(*
---Control step base interface
*)
FUNCTION_BLOCK ActStepBase IMPLEMENTS ITFActStep
VAR CONSTANT
	{attribute 'hide'}
	BEGIN_STEP		:DINT:=10;
	{attribute 'hide'}
	DONE_STEP		:DINT:=60000;
	{attribute 'hide'}
	ERR_DONE_STEP	:DINT:=65000;
	{attribute 'hide'}
	PAUSE_STEP		:DINT:=65500;
END_VAR
VAR_INPUT
END_VAR
VAR_OUTPUT
	step			:DINT;
	errStep			:DINT;
	pauseNextStep	:DINT;
END_VAR
VAR
	//{attribute 'hide'}
	actState		:ST_ActStep_State;
END_VAR

getStep();

(*
---Continue action
*)
METHOD Act_Continue : BOOL
VAR_INPUT
END_VAR
actState.paused:=FALSE;
actState.step:=actState.nextStep;
END_METHOD

(*
---Trigger action
*)
METHOD Act_Ex : BOOL
VAR_INPUT
END_VAR
IF NOT actState.busy AND NOT actState.error THEN
	Act_Ex:=actState.ex:=actState.busy:=TRUE;
ELSE
	Act_Ex:=FALSE;
END_IF
END_METHOD

(*
---Init all status
*)
METHOD Act_Init : BOOL
VAR_INPUT
END_VAR
actState.ex:=actState.pause:=actState.busy:=actState.done:=actState.error:=FALSE;
actState.step:=actState.errStep:=step:=0;
actState.errID:=0;
actState.errMsg:='';

Act_Init:=TRUE;
END_METHOD

(*
---Pause action
*)
METHOD Act_Pause : BOOL
VAR_INPUT
	pause:BOOL;
END_VAR
actState.pause:=pause;
Act_Pause:=TRUE;
END_METHOD

(*
---: add step;
---:
	nextStep: step 增量值;
	checkPause: 是否检测当前 pause; 如果 checkPause:=TRUE, 且暂停被触发后, 当前 step 暂停递增;
*)
METHOD addStep : DINT
VAR_INPUT
	nextStep			:DINT:=0;
	checkPause			:BOOL:=FALSE;// 检查是否暂停，暂停则不递增step
END_VAR
IF checkPause THEN
	IF NOT actState.pause THEN
		actState.step:=actState.step+nextStep;
	END_IF
ELSE
	actState.step:=actState.step+nextStep;
END_IF

addStep:=step:=actState.step;
END_METHOD

(*
---Get action state
*)
METHOD getActState : ST_ActStep_State
VAR_INPUT
END_VAR
getActState:=actState;
END_METHOD

(*
---Get error id
*)
METHOD getErrID : DINT
VAR_INPUT
END_VAR
getErrID:=actState.errID;
END_METHOD

(*
---Get error message
*)
METHOD getErrMsg : STRING(255)
VAR_INPUT
END_VAR
getErrMsg:=actState.errMsg;
END_METHOD

(*
---Get error step
*)
METHOD getErrStep : DINT
VAR_INPUT
END_VAR
getErrStep:=actState.errStep;
END_METHOD

(*
---Get step
*)
METHOD getStep : DINT
VAR_INPUT
END_VAR
getStep:=step:=actState.step;
END_METHOD

(*
---Check busy state
*)
METHOD isBusy : BOOL
VAR_INPUT
END_VAR

isBusy:=actState.busy;
END_METHOD

(*
---Check done state
*)
METHOD isDone : BOOL
VAR_INPUT
END_VAR

isDone:=actState.done;
END_METHOD

(*
---Check error state
*)
METHOD isError : BOOL
VAR_INPUT
END_VAR

isError:=actState.error;
END_METHOD

(*
---Check trigger state
*)
METHOD isEx : BOOL
VAR_INPUT
END_VAR

isEx:=actState.ex;
END_METHOD

(*
---Check pause state
*)
METHOD isPause : BOOL
VAR_INPUT
END_VAR

isPause:=actState.pause;
END_METHOD

(*
---Set busy flag
*)
METHOD setBusyFlag
VAR_INPUT
END_VAR
//actState.busy:=TRUE;
actState.ex:=actState.done:=actState.error:=FALSE;
actState.errID:=0;
actState.step:=step:=actState.errStep:=errStep:=actState.nextStep:=pauseNextStep:=0;
actState.errMsg:='';
END_METHOD

(*
---Set done flag
*)
METHOD setDoneFlag
VAR_INPUT
END_VAR
actState.busy:=FALSE;
actState.pause:=FALSE;
actState.done:=TRUE;
actState.error:=FALSE;
actState.errID:=0;
actState.errMsg:='';
END_METHOD

(*
---Set error done flag
*)
METHOD setErrDoneFlag
VAR_INPUT
END_VAR
actState.busy:=FALSE;
actState.pause:=FALSE;
actState.done:=FALSE;
actState.error:=TRUE;
END_METHOD

(*
---Set error id
*)
METHOD setErrID
VAR_INPUT
	errID:DINT;
END_VAR
actState.errID:=errID;
errStep:=actState.errStep:=actState.step;
END_METHOD

(*
---Set error message
*)
METHOD setErrMsg
VAR_INPUT
	errMsg:STRING(255);
END_VAR
actState.errMsg:=errMsg;
errStep:=actState.errStep:=actState.step;
END_METHOD

(*
---Set error id and error message
*)
METHOD setError
VAR_INPUT
	errID:DINT;
	errMsg:STRING(255);
END_VAR
setErrID(errID);
setErrMsg(errMsg);
END_METHOD

(*
---Go to step:=BEGIN_STEP, BEGIN_STEP is 10;
*)
METHOD toBeginStep : DINT
VAR_INPUT
END_VAR
toBeginStep:=step:=actState.step:=BEGIN_STEP;
END_METHOD

(*
---Go to step:=DONE_STEP, DONE_STEP is 60000;
*)
METHOD toDoneStep : DINT
VAR_INPUT
END_VAR
toDoneStep:=step:=actState.step:=DONE_STEP;
END_METHOD

(*
---Go to step:=ERR_DONE_STEP, ERR_DONE_STEP is 65000;
*)
METHOD toErrDoneStep : DINT
VAR_INPUT
END_VAR
errStep:=actState.errStep:=actState.step;
toErrDoneStep:=step:=actState.step:=ERR_DONE_STEP;
END_METHOD

(*
---Go to pause step:=PAUSE_STEP, PAUSE_STEP is 65500; 
---: nextStep: 从暂停解除之后的下一个step值; 
*)
METHOD toPauseStep : DINT
VAR_INPUT
	nextStep			:DINT:=0;
END_VAR
actState.paused:=TRUE;
actState.nextStep:=pauseNextStep:=nextStep;
actState.step:=PAUSE_STEP;
END_METHOD

(*
---: Go to target step;
---:
	nextStep: step 目标值;
	checkPause: 是否检测当前 pause; 如果 checkPause:=TRUE, 且暂停被触发后, 当前 step 暂停递增;
*)
METHOD toStep : DINT
VAR_INPUT
	nextStep			:DINT:=0;// 跳转到目标step
	checkPause			:BOOL:=FALSE;// 检查是否暂停，暂停则不递增step
END_VAR
IF checkPause THEN
	IF NOT actState.pause THEN
		actState.step:=nextStep;
	END_IF
ELSE
	actState.step:=nextStep;
END_IF

toStep:=step:=actState.step;
END_METHOD

(*
---Go to step:=0;
*)
METHOD toZeroStep : DINT
VAR_INPUT
END_VAR
toZeroStep:=step:=actState.step:=0;
END_METHOD

END_FUNCTION_BLOCK

(* stored: Version 1.1.0.1, ProductVersion 3.1.4024.4
   POU ActStepBase: Id {a3b05ce9-b0d8-4901-8334-9b364782f99a}, SpecialFunc None
   Folder Get: Id {c3272e03-5a93-4152-b0ae-6168d16f9797}
   Folder Is: Id {e5321c25-63a5-402e-adfe-5d46ee6cd96e}
   Folder Set: Id {1ab335a3-1fc3-4c13-b036-90b6f9cd450c}
   Folder Step: Id {6246289c-708c-40ee-87af-f09e5c5a6a94}
   Method Act_Continue: Id {685e1715-541f-48cc-a5a8-aeb8ceb478a8}
   Method Act_Ex: Id {ee5d426f-c21c-4588-9cd1-041b516129ab}
   Method Act_Init: Id {bc88da5d-1db5-4172-84d0-0c4a4812e0bc}
   Method Act_Pause: Id {65e7c203-9edf-43ab-8d51-8fb169bf1513}
   Method addStep: Id {a3a7967b-d647-4f00-99a7-8c408b298864}
   Method getActState: Id {1a9c0758-2142-462a-acf1-4c4397300007}
   Method getErrID: Id {06dccd74-917a-460c-84d1-568d7de16639}
   Method getErrMsg: Id {3af0f11f-c49b-4f09-83d2-e64e58472a23}
   Method getErrStep: Id {454bce6a-c71f-4b03-a774-278d5fb6e8c6}
   Method getStep: Id {7f50d397-fec5-4f44-92a7-4999efcb34dc}
   Method isBusy: Id {293c7294-c67a-498a-80d1-13f65dedd6ab}
   Method isDone: Id {40be26d7-6251-4127-921d-432a2da2024a}
   Method isError: Id {2a1ac8e6-682c-43a7-9d7b-292dabea85c9}
   Method isEx: Id {175e0c94-0529-4d0f-abbc-3b2b40acc23a}
   Method isPause: Id {f842f542-4714-4d5d-a373-306e2496eab1}
   Method setBusyFlag: Id {bb7cf88f-5b32-48f8-b82c-dcec3dc13cd9}
   Method setDoneFlag: Id {f00863fc-41c9-4659-ba37-092cf34a3734}
   Method setErrDoneFlag: Id {2bca7f90-e288-4a13-8c71-97ea40097ee1}
   Method setErrID: Id {0082a529-dbb8-451c-abd8-489562945352}
   Method setErrMsg: Id {6d5b8272-0d11-42df-b798-652dfb08ddc8}
   Method setError: Id {a23b9e4f-ac29-45fd-969b-36d8f3d7337c}
   Method toBeginStep: Id {0426be86-e782-4d34-ac86-7055fdc50e4e}
   Method toDoneStep: Id {0151039e-596d-4631-ba17-b6f29e4e4a74}
   Method toErrDoneStep: Id {3d0517ad-6265-464e-b899-de41966cf145}
   Method toPauseStep: Id {5645af0d-3f6c-44c0-9339-74a58bc8303b}
   Method toStep: Id {ee085535-10e6-4ef5-b17f-706f6c2ad958}
   Method toZeroStep: Id {47530837-7dca-4201-86a5-53024a47b4c9} *)
